{attribute 'qualified_only'}
VAR_GLOBAL PERSISTENT
	testPeristent: INT;
	test_Struct_Pers : Pers_Struct;
END_VAR

(* stored: Version 1.1.0.1, ProductVersion 3.1.4022.12
   GVL GVL_Pers: Id {8293981e-4e86-4079-9efd-975078ce89cc} *)
